(* IEC 61131-3 sources: com.logicals.lc3.webinar/usRTS_RPMControl_iSOC/src_FB_LIB_SAFE/Convert/DWORD, 4 files *)

(* ---- wDWORD_TO_LWORD.iecst ---- *)
NAMESPACE logicals.web.standard
NAMESPACE convert

/*
 * Function block wrapper for IEC 61131-3 TO_LWORD<br>
 * IN =  input value (DWORD)<br>
 * OUT = IN (LWORD)<br>
 */
FUNCTION_BLOCK wDWORD_TO_LWORD
	{ vNameAlignment:="center"; altName:="DWORD_TO_LWORD"; bgColor:="DodgerBlue"; width:=160; hideIONames; }
	VAR_INPUT
		IN : DWORD;
	END_VAR
	VAR_OUTPUT
		OUT: LWORD;
	END_VAR

	OUT := TO_LWORD(IN:=IN, ENO=>ENO);
END_FUNCTION_BLOCK

END_NAMESPACE
END_NAMESPACE

(* ---- wDWORD_TO_UDINT.iecst ---- *)
NAMESPACE logicals.web.standard
NAMESPACE convert

/*
 * Function block wrapper for IEC 61131-3 TO_UDINT<br>
 * IN =  input value (DWORD)<br>
 * OUT = IN (UDINT)<br>
 */
FUNCTION_BLOCK wDWORD_TO_UDINT
	{ vNameAlignment:="center"; altName:="DWORD_TO_UDINT"; bgColor:="Plum"; width:=140; hideIONames; }
	VAR_INPUT
		IN : DWORD;
	END_VAR
	VAR_OUTPUT
		OUT: UDINT;
	END_VAR

	OUT := TO_UDINT(IN:=IN, ENO=>ENO);
END_FUNCTION_BLOCK

END_NAMESPACE
END_NAMESPACE

(* ---- wTRUNC_DWORD_TO_BYTE.iecst ---- *)
NAMESPACE logicals.web.standard
NAMESPACE convert

/*
 * Function block wrapper for IEC 61131-3 TO_BYTE<br>
 * IN =  input value (DWORD)<br>
 * OUT = IN (BYTE)<br>
 */
FUNCTION_BLOCK wTRUNC_DWORD_TO_BYTE
	{ vNameAlignment:="center"; altName:="TRUNC_DWORD_TO_BYTE"; bgColor:="DodgerBlue"; width:=200; hideIONames; }
	VAR_INPUT
		IN : DWORD;
	END_VAR
	VAR_OUTPUT
		OUT: BYTE;
	END_VAR

	OUT := TO_BYTE(IN:=IN, ENO=>ENO);
END_FUNCTION_BLOCK

END_NAMESPACE
END_NAMESPACE

(* ---- wTRUNC_DWORD_TO_WORD.iecst ---- *)
NAMESPACE logicals.web.standard
NAMESPACE convert

/*
 * Function block wrapper for IEC 61131-3 TO_WORD<br>
 * IN =  input value (DWORD)<br>
 * OUT = IN (WORD)<br>
 */
FUNCTION_BLOCK wTRUNC_DWORD_TO_WORD
	{ vNameAlignment:="center"; altName:="TRUNC_DWORD_TO_WORD"; bgColor:="DodgerBlue"; width:=200; hideIONames; }
	VAR_INPUT
		IN : DWORD;
	END_VAR
	VAR_OUTPUT
		OUT: WORD;
	END_VAR

	OUT := TO_WORD(IN:=IN, ENO=>ENO);
END_FUNCTION_BLOCK

END_NAMESPACE
END_NAMESPACE
